FUNCTION_BLOCK FB_ModeCBox IMPLEMENTS I_Mode
VAR_INPUT
END_VAR
VAR_OUTPUT
END_VAR
VAR
END_VAR

METHOD Auto
VAR_INPUT
	bEnable : BOOL;
END_VAR
IF bEnable THEN 
	Output.eMode := E_Mode.Auto;
END_IF
END_METHOD

METHOD Manual
VAR_INPUT
	bEnable : BOOL;
END_VAR
IF bEnable THEN 
	Output.eMode := E_Mode.Manual;
END_IF
END_METHOD

METHOD OFF 
VAR_INPUT
	bEnable : BOOL;
END_VAR
IF bEnable THEN 
	Output.eMode := E_Mode.OFF;
END_IF
END_METHOD

END_FUNCTION_BLOCK

(* stored: Version 1.1.0.1, ProductVersion 3.1.4024.12
   POU FB_ModeCBox: Id {507e1aeb-a33b-4800-85b4-509438143db2}, SpecialFunc None
   Method Auto: Id {1b9c99d4-5e07-4a51-9eba-e425764ec612}
   Method Manual: Id {6268042c-94fe-4f98-8dd7-0c72f90927b3}
   Method OFF: Id {9b9adc2b-14e0-4047-90a5-5b93f9d701dc} *)
